FUNCTION_BLOCK DummyControl (* Basic Function Block Type *)
  (* Standard: 61499-2 *)
  (* Version 0.0, 6/17/2016, Andrei, nxtControl GmbH, Template *)
  PACKAGE Main;
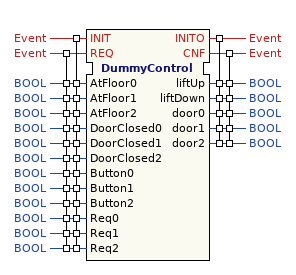
  EVENT_INPUT
    INIT WITH AtFloor0, AtFloor1, AtFloor2, DoorClosed0, DoorClosed1, DoorClosed2, Button0, Button1, Button2, Req0, Req1, Req2; (* Initialization Request *)
    REQ WITH AtFloor0, AtFloor1, AtFloor2, DoorClosed0, DoorClosed1, DoorClosed2, Button0, Button1, Button2, Req0, Req1, Req2; (* Normal Execution Request *)
  END_EVENT
  EVENT_OUTPUT
    INITO WITH liftUp, liftDown, door0, door1, door2; (* Initialization Confirm *)
    CNF WITH liftUp, liftDown, door0, door1, door2; (* Execution Confirmation *)
  END_EVENT
  VAR_INPUT
    AtFloor0 : BOOL; (* Input event qualifier *)
    AtFloor1 : BOOL;
    AtFloor2 : BOOL;
    DoorClosed0 : BOOL;
    DoorClosed1 : BOOL;
    DoorClosed2 : BOOL;
    Button0 : BOOL;
    Button1 : BOOL;
    Button2 : BOOL;
    Req0 : BOOL;
    Req1 : BOOL;
    Req2 : BOOL;
  END_VAR
  VAR_OUTPUT
    liftUp : BOOL;
    liftDown : BOOL; (* Output event qualifier *)
    door0 : BOOL;
    door1 : BOOL;
    door2 : BOOL;
  END_VAR
  VAR
    AtSomeFloor : BOOL;
    IsRequested : BOOL;
    NeedStop : BOOL;
  END_VAR
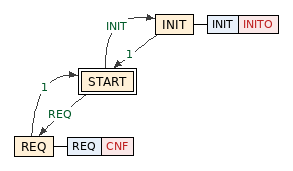
  EC_STATES
    START; (* Initial State *)
    INIT : INIT -> INITO; (* Initialization *)
    REQ : REQ -> CNF; (* Normal execution *)
  END_STATES
  EC_TRANSITIONS
    START TO INIT := INIT;
    INIT TO START := 1;
    START TO REQ := REQ;
    REQ TO START := 1;
  END_TRANSITIONS
  ALGORITHM INIT IN ST: (* Initialization algorithm *)
liftDown := TRUE;
  END_ALGORITHM
  ALGORITHM REQ IN ST: (* Normally executed algorithm *)
AtSomeFloor := AtFloor0 OR AtFloor1 OR AtFloor2;
IsRequested := (Button0 OR Req0) OR (Button1 OR Req1) OR (Button2 OR Req2);
NeedStop := FALSE;

(* Close door if opened *)
IF NOT DoorClosed0 THEN door0 := FALSE; END_IF;
IF NOT DoorClosed1 THEN door1 := FALSE; END_IF;
IF NOT DoorClosed2 THEN door2 := FALSE; END_IF;

(* Doesn't change direction while moving *)
IF AtSomeFloor THEN
	(* Stop if nowhere to go *)
	IF NOT IsRequested THEN
		liftUp := FALSE;
		liftDown := FALSE;
	ELSE
		IF NOT (DoorClosed0 AND DoorClosed1 AND DoorClosed2) THEN
			NeedStop := TRUE;
		END_IF;
		(* Check if we arrived on one of the requested floors (if true, open a door) *)
		IF AtFloor0 AND (Button0 OR Req0) THEN
			door0 := TRUE;
			NeedStop := TRUE;
		END_IF;
		IF AtFloor1 AND (Button1 OR Req1) THEN
			door1 := TRUE;
			NeedStop := TRUE;
		END_IF;
		IF AtFloor2 AND (Button2 OR Req2) THEN
			door2 := TRUE;
			NeedStop := TRUE;
		END_IF;
		(* If arrived on the right floor, stop *)
		IF NeedStop THEN
  		liftUp := FALSE;
	  	liftDown := FALSE;
	  ELSE
	  	(* 0 floor requeted - go down *)
	  	IF (Button0 OR Req0) THEN
    		liftUp := FALSE;
	    	liftDown := TRUE;
	  	END_IF;
	  	(* 2 floor requeted - go up *)
	  	IF (Button2 OR Req2) THEN
    		liftUp := TRUE;
	    	liftDown := FALSE;
	  	END_IF;
	  	(* Check if we are lower or higher *)
	  	IF (Button1 OR Req1) THEN
	  		liftUp := AtFloor0;
	  		liftDown := AtFloor2;
	  	END_IF;
	  END_IF;
	END_IF;
END_IF;
  END_ALGORITHM
END_FUNCTION_BLOCK
